// TIA Portal V21 export
ORGANIZATION_BLOCK "Main"   // OB1, LAD, ProgramCycle
TITLE = "Main Program Sweep (Cycle)"
{ S7_Optimized_Access := 'TRUE' }
// stored: SetENOAutomatically false
   VAR_INPUT
      Initial_Call : Bool;   // Initial call of this OB
      Remanence : Bool;   // =True, if remanent data are available
   END_VAR
BEGIN

REGION Network 1
   // Start Stop motor
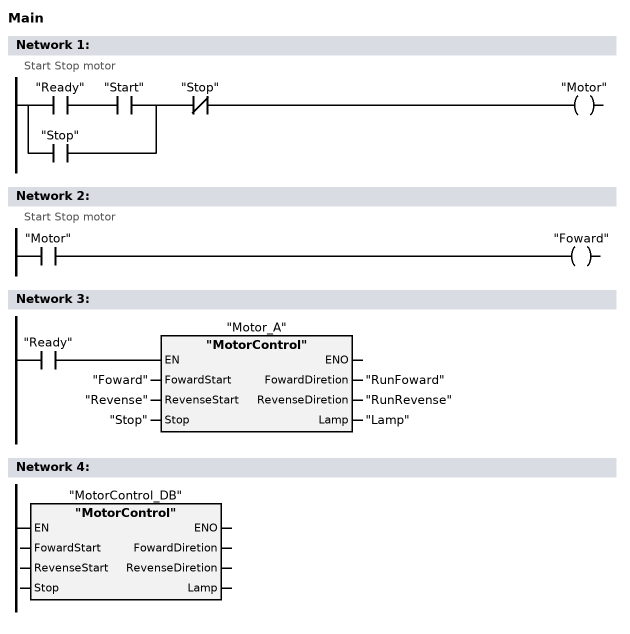
   RUNG wire#powerrail
      Contact( "Ready" )
      Contact( "Start" )
      wire#w1
      I_Contact( "Stop" )
      Coil( "Motor" )
   END_RUNG
   RUNG wire#powerrail
      Contact( "Stop" )
   END_RUNG wire#w1
   // the same network as SCL:
   "Motor" := (("Ready" AND "Start") OR "Stop") AND NOT "Stop";
END_REGION

REGION Network 2
   // Start Stop motor
   RUNG wire#powerrail
      Contact( "Motor" )
      Coil( "Foward" )
   END_RUNG
   // the same network as SCL:
   "Foward" := "Motor";
END_REGION

REGION Network 3
   RUNG wire#powerrail
      Contact( "Ready" )
      "Motor_A"(FowardStart := "Foward", RevenseStart := "Revense", Stop := "Stop", FowardDiretion => "RunFoward", RevenseDiretion => "RunRevense", Lamp => "Lamp")
   END_RUNG
   // the same network as SCL:
   IF "Ready" THEN
       "Motor_A"(FowardStart := "Foward",   // "MotorControl"
                 RevenseStart := "Revense",
                 Stop := "Stop",
                 FowardDiretion => "RunFoward",
                 RevenseDiretion => "RunRevense",
                 Lamp => "Lamp");
   END_IF;
END_REGION

REGION Network 4
   RUNG wire#powerrail
      "MotorControl_DB"(FowardStart :=, RevenseStart :=, Stop :=, FowardDiretion =>, RevenseDiretion =>, Lamp =>)
   END_RUNG
   // the same network as SCL:
   "MotorControl_DB"();   // "MotorControl"
END_REGION
END_ORGANIZATION_BLOCK
